FUNCTION TryConvert_DT_TO_LWORD : BOOL
VAR_INPUT
	in : DT;
	out : REFERENCE TO LWORD;
END_VAR

out := DT_TO_LWORD(in);
TryConvert_DT_TO_LWORD := TRUE;

END_FUNCTION

(* stored: Version 1.1.0.1, ProductVersion 3.1.4024.12
   POU TryConvert_DT_TO_LWORD: Id {a950b503-a5db-4f3e-9504-f71978ddcf4d}, SpecialFunc None *)
